(* Logix 5000 project; controller Thurs_Lab2 vendor 1 type 14 code 156 rev 30.11; software revision 30.00; part 4 of 5 *)
(* tags used below, declared in another part *)
   STEP1 : SFC_STEP;
   A_VFD_RUN : BOOL;
   AUTO : BOOL;
   AVERAGE : DINT;
   BLUE_STACK_LITE : BOOL;
   COUNTER : COUNTER;
   CYCLE_COUNT : COUNTER;
   CYCLE_TIME : TIMER;
   CYL1_EXT_4_SORTING : BOOL;
   CYL1_EXT_PX : BOOL;
   CYL1_RET_4_SORTING : BOOL;
   CYL1_RET_PX : BOOL;
   CYL2_EXT_4_SORTING : BOOL;
   CYL2_EXT_PX : BOOL;
   CYL3_EXT : BOOL;
   CYL3_RET : BOOL;
   CYL4_EXT : BOOL;
   CYLINDER1_EXTEND : BOOL;
   CYLINDER1_RETRACT : BOOL;
   CYLINDER2_EXTEND : BOOL;
   CYLINDERSTATUS : DINT;
   DEEP : COUNTER;
   DELAY_PE_INPUT_PSW : TIMER;
   DELAY_PE_INPUT_STATE : TIMER;
   DRILL3 : DRILL3;
   DRILL4 : DRILL4;
   EXTEND : TIMER;
   FAULT : BOOL;
   FAULT_COUNTER : COUNTER;
   GREEN_STACK_LITE : BOOL;
   LAST_CYCLE_COUNT : COUNTER;
   LAST_CYCLE_TIME : DINT;
   MOTOR_WHEEL : BOOL;
   MOTOR_WHEEL_PE : BOOL;
   ONE_SHOT_PSW0 : BOOL;
   ONE_SHOT_PSW1 : BOOL;
   ONE_SHOT_STATE0 : BOOL;
   ONE_SHOT_STATE1 : BOOL;
   OP3_STOP : BOOL;
   OP4_STOP : BOOL;
   OP7_STOP : BOOL;
   OPERATION : DINT;
   OPERATION_7_OVER : BOOL;
   OPERATION_7_REJECT : BOOL;
   OPERATION_7_UNDER : BOOL;
   OPERATION_DONE : DINT;
   OPERATION_OFF : DINT;
   OUTPUT : INT;
   PARTS : COUNTER;
   PARTS_COUNT_TOTALIZER : COUNTER;
   PB1 : BOOL;
   PB1_ON : DINT;
   PILOT_LIGHT_0 : BOOL;
   PILOT_LIGHT_1 : BOOL;
   PILOT_LIGHT_2 : BOOL;
   PILOT_LIGHT_3 : BOOL;
   PILOT_LIGHT_4 : BOOL;
   PILOT_LIGHT_5 : BOOL;
   PREVENT_FAULT_7 : DINT;
   PRODUCTION_ONE_SHOT : BOOL;
   PV_FAULT_COUNT_RESET : BOOL;
   PV_FAULT_RESET : BOOL;
   PV_LAST_CYCLE_TIME1 : DINT;
   PV_LAST_CYCLE_TIME2 : DINT;
   PV_LAST_CYCLE_TIME3 : DINT;
   PV_LAST_CYCLE_TIME4 : DINT;
   PV_LAST_CYCLE_TIME5 : DINT;
   PV_MAX_DEPTH : DINT;
   PV_MIN_DEPTH : DINT;
   PV_PARTS_COUNT_RESET : BOOL;
   PV_RESET : BOOL;
   RED_STACK_LITE : BOOL;
   RESET : BOOL;
   REVOLUTIONS : COUNTER;
   RUN_DC_MOTOR : BOOL;
   SEQ_A_TO_D_COMPLETE : BOOL;
   SEQ_EN : BOOL;
   SETSPEED7 : DINT;
   SHALLOW : COUNTER;
   SORT_SEQ_FOR_REJECT : DINT;
   STA : DINT;
   START_SIGNAL : BOOL;
   STATE : DINT;
   STEP : DINT;
   T : DINT;
   Timer : TIMER;
   TIMER_CELL_DONE : TIMER;
   TO_CELL : TO_CELL;
   TOO_DEEP : BOOL;
   TOO_SHALLOW : BOOL;
   TRANSFER7 : TIMER;
   UP2SPEED7 : TIMER;
   WHITE_STACK_LITE : BOOL;
   YELLOW_STACK_LITE : BOOL;
   ZEROSPEED7 : TIMER;
(* MainProgram, continued *)

ROUTINE OP3_DRILL_PSW   (* ladder *)
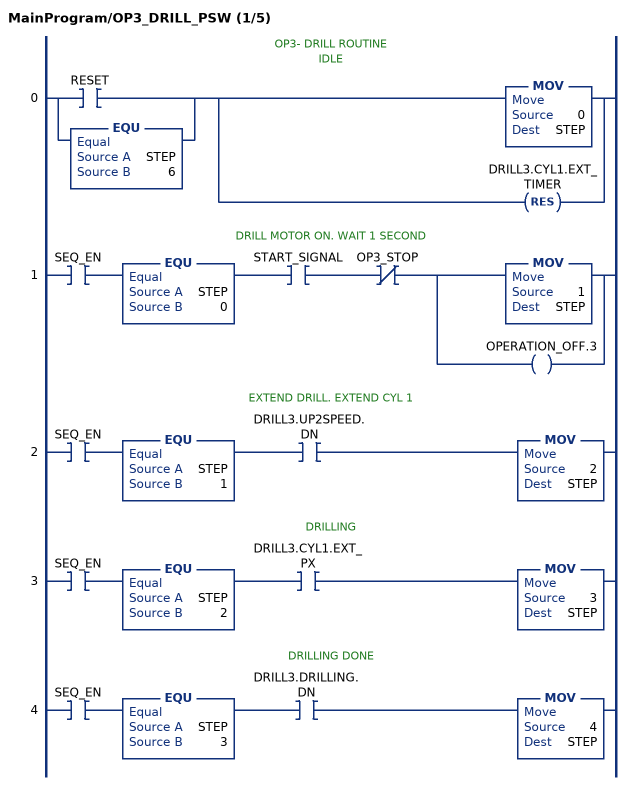
   // OP3- DRILL ROUTINE
   // IDLE
   0: [XIC(RESET) ,EQU(STEP,6) ][MOV(0,STEP) ,RES(DRILL3.CYL1.EXT_TIMER) ];
   // DRILL MOTOR ON. WAIT 1 SECOND
   1: XIC(SEQ_EN)EQU(STEP,0)XIC(START_SIGNAL)XIO(OP3_STOP)[MOV(1,STEP) ,OTE(OPERATION_OFF.3) ];
   // EXTEND DRILL. EXTEND CYL 1
   2: XIC(SEQ_EN)EQU(STEP,1)XIC(DRILL3.UP2SPEED.DN)MOV(2,STEP);
   // DRILLING
   3: XIC(SEQ_EN)EQU(STEP,2)XIC(DRILL3.CYL1.EXT_PX)MOV(3,STEP);
   // DRILLING DONE
   4: XIC(SEQ_EN)EQU(STEP,3)XIC(DRILL3.DRILLING.DN)MOV(4,STEP);
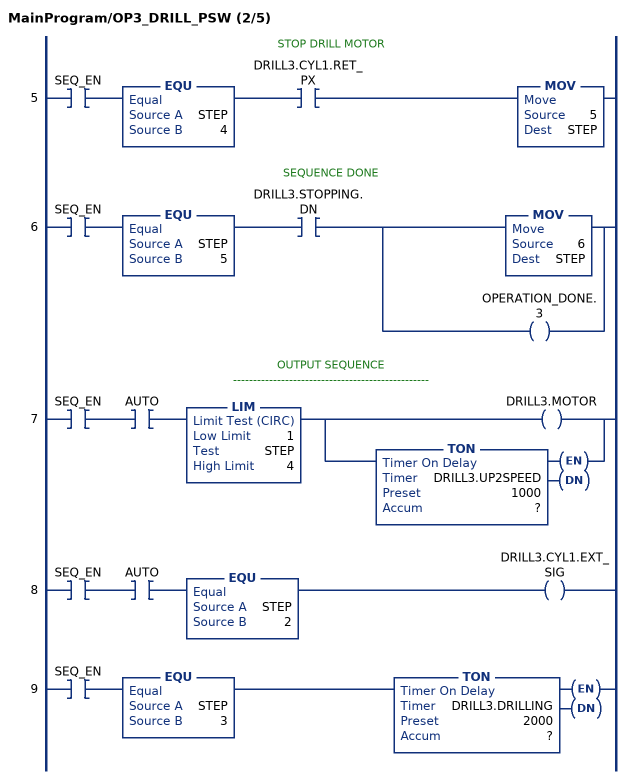
   // STOP DRILL MOTOR
   5: XIC(SEQ_EN)EQU(STEP,4)XIC(DRILL3.CYL1.RET_PX)MOV(5,STEP);
   // SEQUENCE DONE
   6: XIC(SEQ_EN)EQU(STEP,5)XIC(DRILL3.STOPPING.DN)[MOV(6,STEP) ,OTE(OPERATION_DONE.3) ];
   // OUTPUT SEQUENCE
   // -------------------------------------------------
   7: XIC(SEQ_EN)XIC(AUTO)LIM(1,STEP,4)[OTE(DRILL3.MOTOR) ,TON(DRILL3.UP2SPEED,?,?) ];
   8: XIC(SEQ_EN)XIC(AUTO)EQU(STEP,2)OTE(DRILL3.CYL1.EXT_SIG);
   9: XIC(SEQ_EN)EQU(STEP,3)TON(DRILL3.DRILLING,?,?);
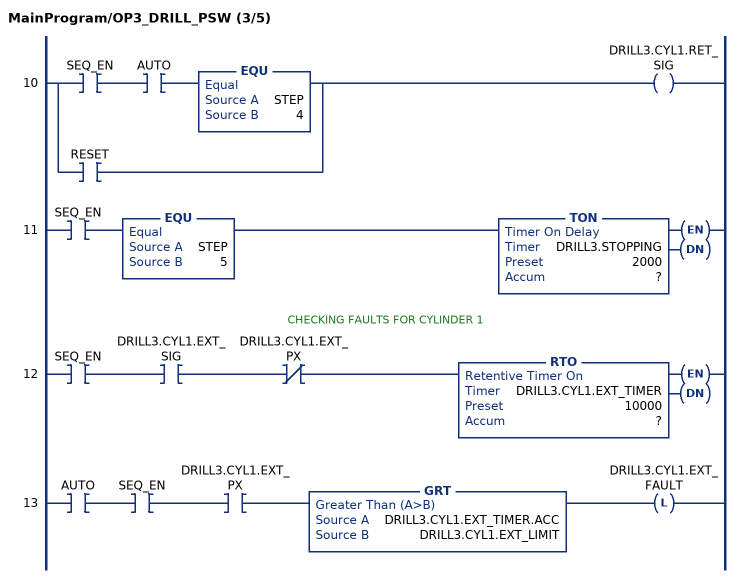
   10: [XIC(SEQ_EN) XIC(AUTO) EQU(STEP,4) ,XIC(RESET) ]OTE(DRILL3.CYL1.RET_SIG);
   11: XIC(SEQ_EN)EQU(STEP,5)TON(DRILL3.STOPPING,?,?);
   // CHECKING FAULTS FOR CYLINDER 1
   12: XIC(SEQ_EN)XIC(DRILL3.CYL1.EXT_SIG)XIO(DRILL3.CYL1.EXT_PX)RTO(DRILL3.CYL1.EXT_TIMER,?,?);
   13: XIC(AUTO)XIC(SEQ_EN)XIC(DRILL3.CYL1.EXT_PX)GRT(DRILL3.CYL1.EXT_TIMER.ACC,DRILL3.CYL1.EXT_LIMIT)OTL(DRILL3.CYL1.EXT_FAULT);
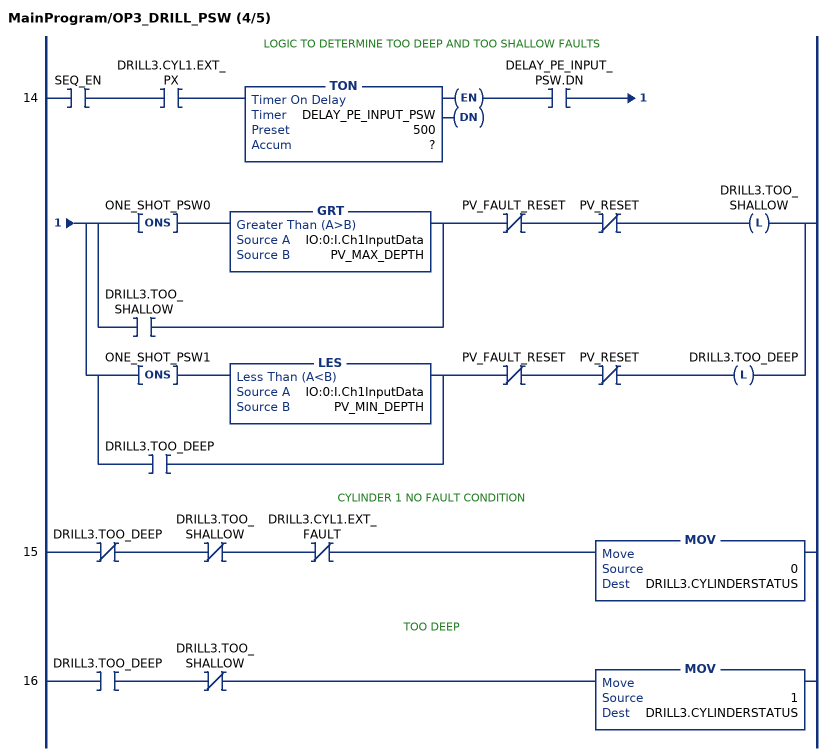
   // LOGIC TO DETERMINE TOO DEEP AND TOO SHALLOW FAULTS
   14: XIC(SEQ_EN)XIC(DRILL3.CYL1.EXT_PX)TON(DELAY_PE_INPUT_PSW,?,?)XIC(DELAY_PE_INPUT_PSW.DN)[[ONS(ONE_SHOT_PSW0) GRT(IO:0:I.Ch1InputData,PV_MAX_DEPTH) ,XIC(DRILL3.TOO_SHALLOW) ] XIO(PV_FAULT_RESET) XIO(PV_RESET) OTL(DRILL3.TOO_SHALLOW) ,[ONS(ONE_SHOT_PSW1) LES(IO:0:I.Ch1InputData,PV_MIN_DEPTH) ,XIC(DRILL3.TOO_DEEP) ] XIO(PV_FAULT_RESET) XIO(PV_RESET) OTL(DRILL3.TOO_DEEP) ];
   // CYLINDER 1 NO FAULT CONDITION
   15: XIO(DRILL3.TOO_DEEP)XIO(DRILL3.TOO_SHALLOW)XIO(DRILL3.CYL1.EXT_FAULT)MOV(0,DRILL3.CYLINDERSTATUS);
   // TOO DEEP
   16: XIC(DRILL3.TOO_DEEP)XIO(DRILL3.TOO_SHALLOW)MOV(1,DRILL3.CYLINDERSTATUS);
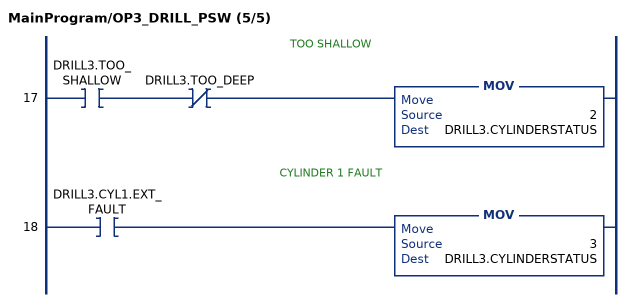
   // TOO SHALLOW
   17: XIC(DRILL3.TOO_SHALLOW)XIO(DRILL3.TOO_DEEP)MOV(2,DRILL3.CYLINDERSTATUS);
   // CYLINDER 1 FAULT
   18: XIC(DRILL3.CYL1.EXT_FAULT)MOV(3,DRILL3.CYLINDERSTATUS);
END_ROUTINE

ROUTINE OP4_DRILL_STATE   (* ladder *)
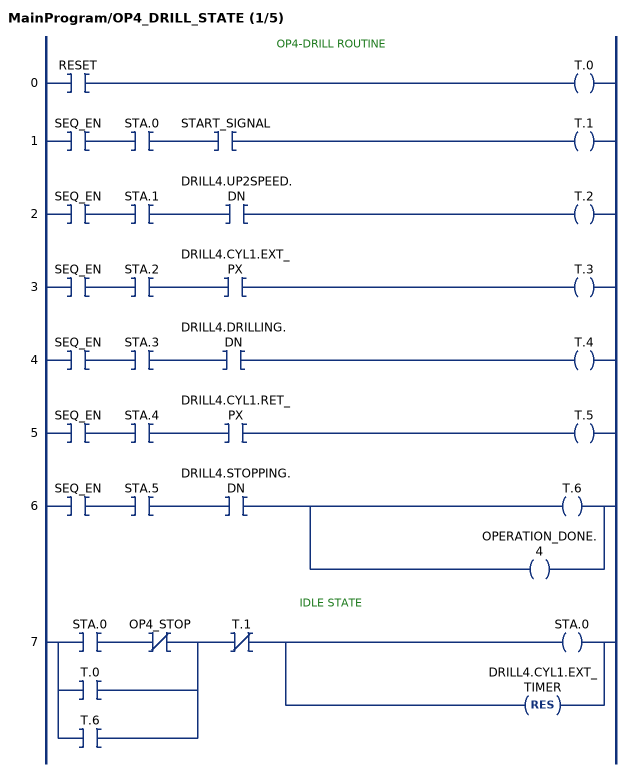
   // OP4-DRILL ROUTINE
   0: XIC(RESET)OTE(T.0);
   1: XIC(SEQ_EN)XIC(STA.0)XIC(START_SIGNAL)OTE(T.1);
   2: XIC(SEQ_EN)XIC(STA.1)XIC(DRILL4.UP2SPEED.DN)OTE(T.2);
   3: XIC(SEQ_EN)XIC(STA.2)XIC(DRILL4.CYL1.EXT_PX)OTE(T.3);
   4: XIC(SEQ_EN)XIC(STA.3)XIC(DRILL4.DRILLING.DN)OTE(T.4);
   5: XIC(SEQ_EN)XIC(STA.4)XIC(DRILL4.CYL1.RET_PX)OTE(T.5);
   6: XIC(SEQ_EN)XIC(STA.5)XIC(DRILL4.STOPPING.DN)[OTE(T.6) ,OTE(OPERATION_DONE.4) ];
   // IDLE STATE
   7: [XIC(STA.0) XIO(OP4_STOP) ,XIC(T.0) ,XIC(T.6) ]XIO(T.1)[OTE(STA.0) ,RES(DRILL4.CYL1.EXT_TIMER) ];
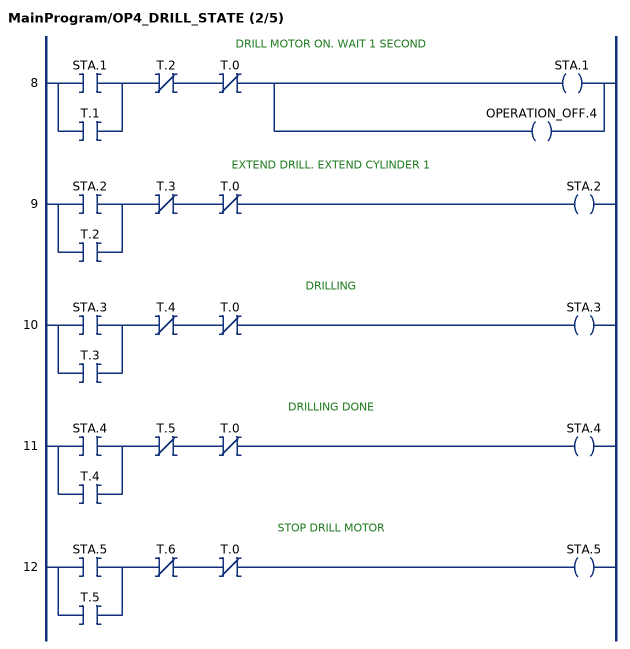
   // DRILL MOTOR ON. WAIT 1 SECOND
   8: [XIC(STA.1) ,XIC(T.1) ]XIO(T.2)XIO(T.0)[OTE(STA.1) ,OTE(OPERATION_OFF.4) ];
   // EXTEND DRILL. EXTEND CYLINDER 1
   9: [XIC(STA.2) ,XIC(T.2) ]XIO(T.3)XIO(T.0)OTE(STA.2);
   // DRILLING
   10: [XIC(STA.3) ,XIC(T.3) ]XIO(T.4)XIO(T.0)OTE(STA.3);
   // DRILLING DONE
   11: [XIC(STA.4) ,XIC(T.4) ]XIO(T.5)XIO(T.0)OTE(STA.4);
   // STOP DRILL MOTOR
   12: [XIC(STA.5) ,XIC(T.5) ]XIO(T.6)XIO(T.0)OTE(STA.5);
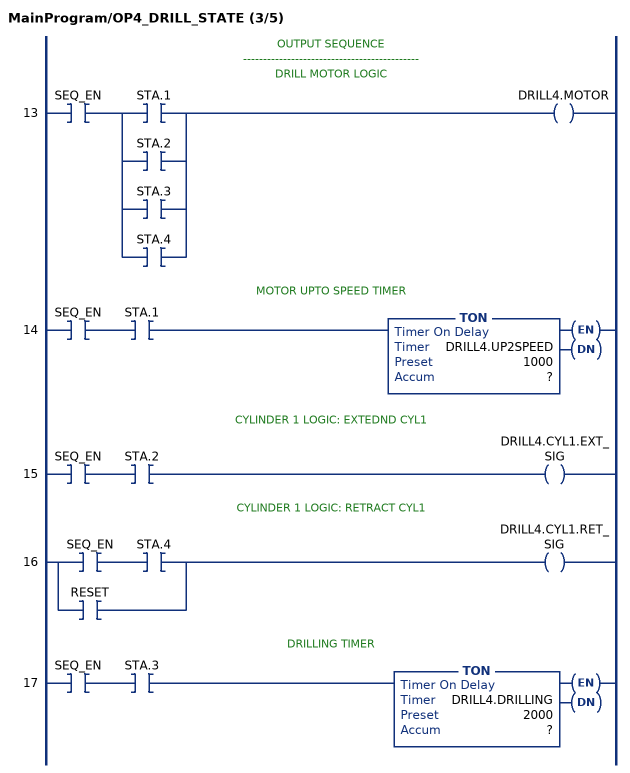
   // OUTPUT SEQUENCE
   // --------------------------------------------
   // DRILL MOTOR LOGIC
   13: XIC(SEQ_EN)[XIC(STA.1) ,XIC(STA.2) ,XIC(STA.3) ,XIC(STA.4) ]OTE(DRILL4.MOTOR);
   // MOTOR UPTO SPEED TIMER
   14: XIC(SEQ_EN)XIC(STA.1)TON(DRILL4.UP2SPEED,?,?);
   // CYLINDER 1 LOGIC: EXTEDND CYL1
   15: XIC(SEQ_EN)XIC(STA.2)OTE(DRILL4.CYL1.EXT_SIG);
   // CYLINDER 1 LOGIC: RETRACT CYL1
   16: [XIC(SEQ_EN) XIC(STA.4) ,XIC(RESET) ]OTE(DRILL4.CYL1.RET_SIG);
   // DRILLING TIMER
   17: XIC(SEQ_EN)XIC(STA.3)TON(DRILL4.DRILLING,?,?);
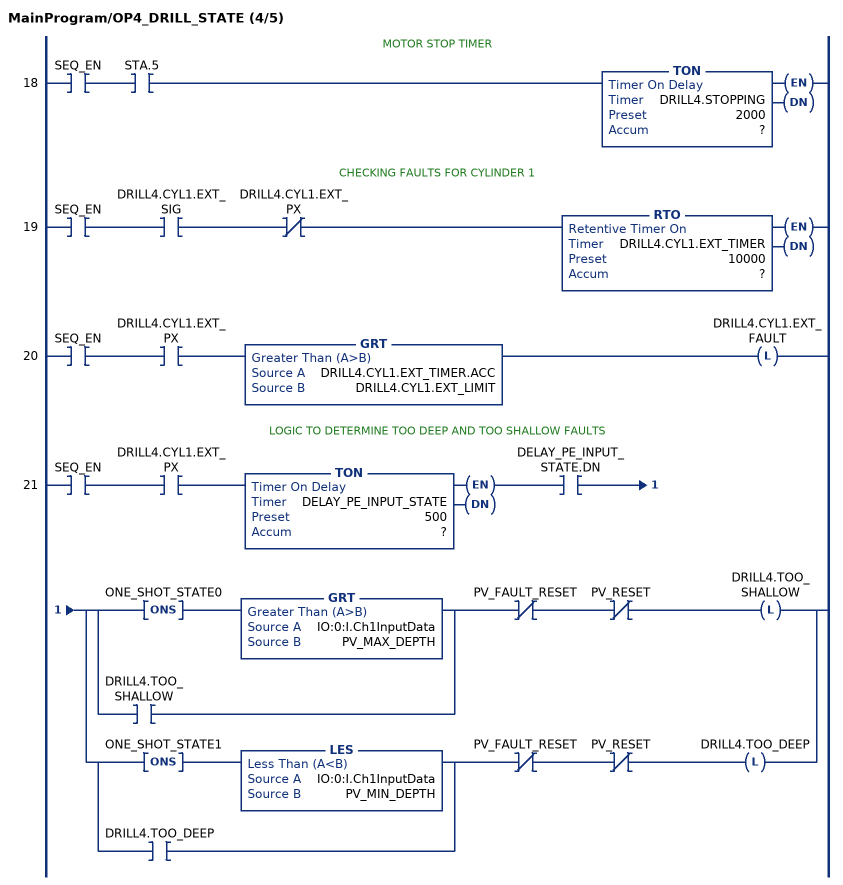
   // MOTOR STOP TIMER
   18: XIC(SEQ_EN)XIC(STA.5)TON(DRILL4.STOPPING,?,?);
   // CHECKING FAULTS FOR CYLINDER 1
   19: XIC(SEQ_EN)XIC(DRILL4.CYL1.EXT_SIG)XIO(DRILL4.CYL1.EXT_PX)RTO(DRILL4.CYL1.EXT_TIMER,?,?);
   20: XIC(SEQ_EN)XIC(DRILL4.CYL1.EXT_PX)GRT(DRILL4.CYL1.EXT_TIMER.ACC,DRILL4.CYL1.EXT_LIMIT)OTL(DRILL4.CYL1.EXT_FAULT);
   // LOGIC TO DETERMINE TOO DEEP AND TOO SHALLOW FAULTS
   21: XIC(SEQ_EN)XIC(DRILL4.CYL1.EXT_PX)TON(DELAY_PE_INPUT_STATE,?,?)XIC(DELAY_PE_INPUT_STATE.DN)[[ONS(ONE_SHOT_STATE0) GRT(IO:0:I.Ch1InputData,PV_MAX_DEPTH) ,XIC(DRILL4.TOO_SHALLOW) ] XIO(PV_FAULT_RESET) XIO(PV_RESET) OTL(DRILL4.TOO_SHALLOW) ,[ONS(ONE_SHOT_STATE1) LES(IO:0:I.Ch1InputData,PV_MIN_DEPTH) ,XIC(DRILL4.TOO_DEEP) ] XIO(PV_FAULT_RESET) XIO(PV_RESET) OTL(DRILL4.TOO_DEEP) ];
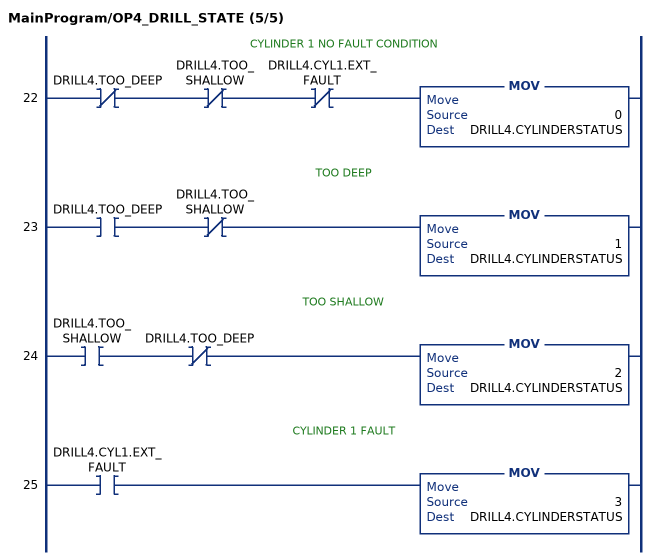
   // CYLINDER 1 NO FAULT CONDITION
   22: XIO(DRILL4.TOO_DEEP)XIO(DRILL4.TOO_SHALLOW)XIO(DRILL4.CYL1.EXT_FAULT)MOV(0,DRILL4.CYLINDERSTATUS);
   // TOO DEEP
   23: XIC(DRILL4.TOO_DEEP)XIO(DRILL4.TOO_SHALLOW)MOV(1,DRILL4.CYLINDERSTATUS);
   // TOO SHALLOW
   24: XIC(DRILL4.TOO_SHALLOW)XIO(DRILL4.TOO_DEEP)MOV(2,DRILL4.CYLINDERSTATUS);
   // CYLINDER 1 FAULT
   25: XIC(DRILL4.CYL1.EXT_FAULT)MOV(3,DRILL4.CYLINDERSTATUS);
END_ROUTINE

ROUTINE OUTPUT_BUFFERING   (* function block diagram *)
   SHEET 1
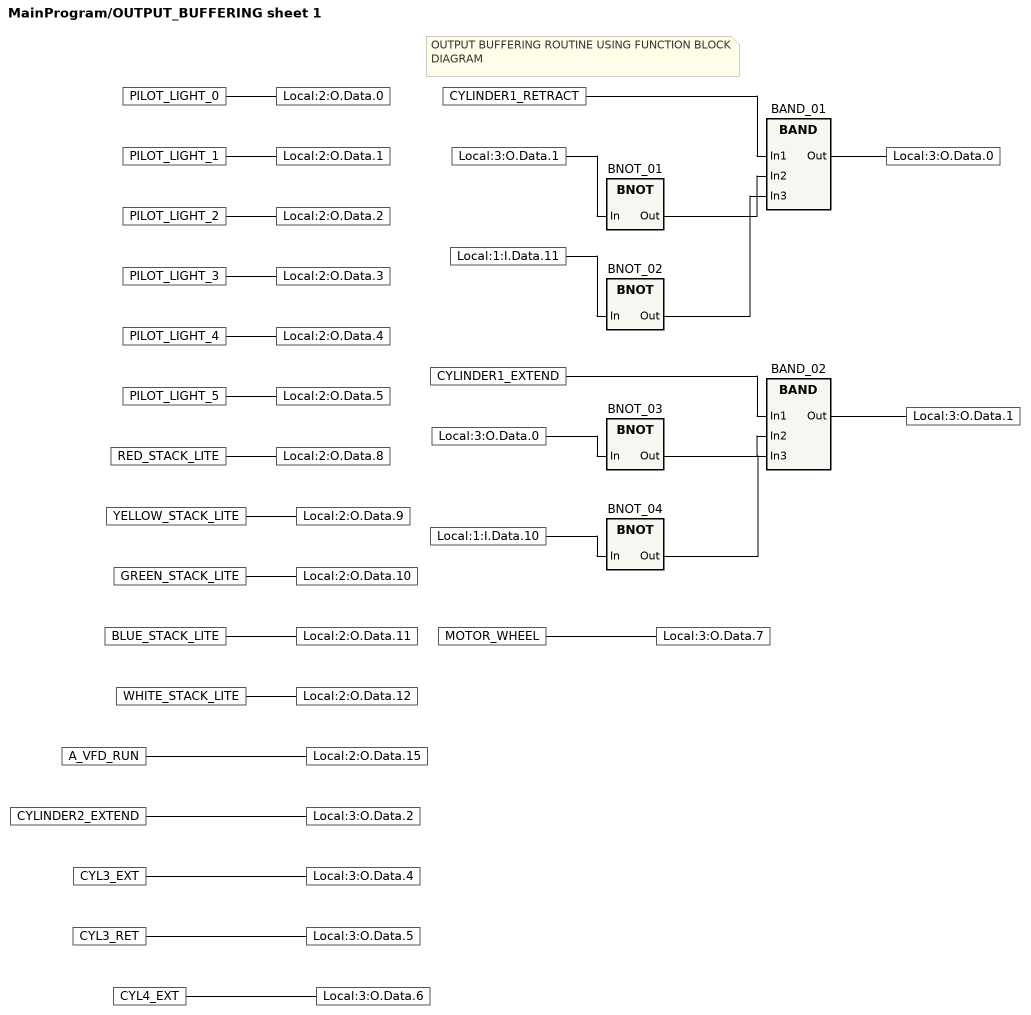
   // OUTPUT BUFFERING ROUTINE USING FUNCTION BLOCK DIAGRAM
   Local:2:O.Data.0 := PILOT_LIGHT_0;
   Local:2:O.Data.1 := PILOT_LIGHT_1;
   Local:2:O.Data.2 := PILOT_LIGHT_2;
   Local:2:O.Data.3 := PILOT_LIGHT_3;
   Local:2:O.Data.4 := PILOT_LIGHT_4;
   Local:2:O.Data.5 := PILOT_LIGHT_5;
   Local:2:O.Data.8 := RED_STACK_LITE;
   Local:2:O.Data.9 := YELLOW_STACK_LITE;
   Local:2:O.Data.10 := GREEN_STACK_LITE;
   Local:2:O.Data.11 := BLUE_STACK_LITE;
   Local:2:O.Data.12 := WHITE_STACK_LITE;
   Local:2:O.Data.15 := A_VFD_RUN;
   Local:3:O.Data.2 := CYLINDER2_EXTEND;
   Local:3:O.Data.4 := CYL3_EXT;
   Local:3:O.Data.5 := CYL3_RET;
   Local:3:O.Data.6 := CYL4_EXT;
   BNOT_01 : BNOT(In := Local:3:O.Data.1);
   BNOT_02 : BNOT(In := Local:1:I.Data.11);
   BNOT_03 : BNOT(In := Local:3:O.Data.0);
   BNOT_04 : BNOT(In := Local:1:I.Data.10);
   Local:3:O.Data.7 := MOTOR_WHEEL;
   BAND_01 : BAND(In1 := CYLINDER1_RETRACT, In2 := BNOT_01.Out, In3 := BNOT_02.Out);
   BAND_02 : BAND(In1 := CYLINDER1_EXTEND, In2 := BNOT_03.Out, In3 := BNOT_04.Out);
   Local:3:O.Data.0 := BAND_01.Out;
   Local:3:O.Data.1 := BAND_02.Out;
END_ROUTINE

ROUTINE PRODUCTION   (* ladder *)
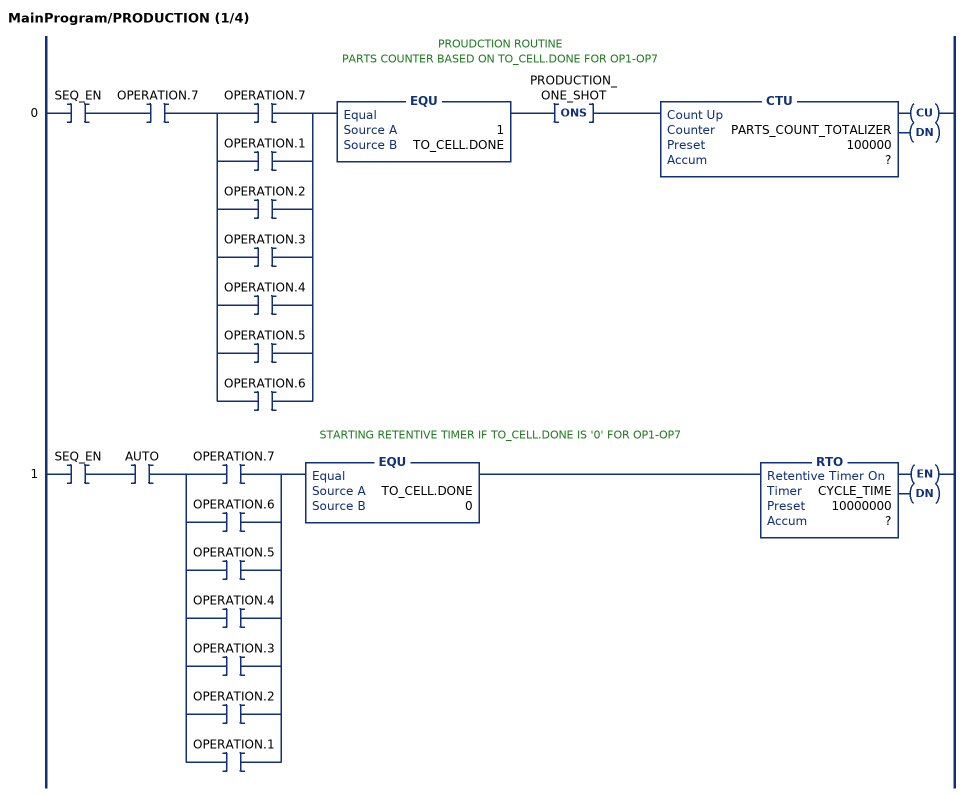
   // PROUDCTION ROUTINE
   // PARTS COUNTER BASED ON TO_CELL.DONE FOR OP1-OP7
   0: XIC(SEQ_EN)XIC(OPERATION.7)[XIC(OPERATION.7) ,XIC(OPERATION.1) ,XIC(OPERATION.2) ,XIC(OPERATION.3) ,XIC(OPERATION.4) ,XIC(OPERATION.5) ,XIC(OPERATION.6) ]EQU(1,TO_CELL.DONE)ONS(PRODUCTION_ONE_SHOT)CTU(PARTS_COUNT_TOTALIZER,?,?);
   // STARTING RETENTIVE TIMER IF TO_CELL.DONE IS '0' FOR OP1-OP7
   1: XIC(SEQ_EN)XIC(AUTO)[XIC(OPERATION.7) ,XIC(OPERATION.6) ,XIC(OPERATION.5) ,XIC(OPERATION.4) ,XIC(OPERATION.3) ,XIC(OPERATION.2) ,XIC(OPERATION.1) ]EQU(TO_CELL.DONE,0)RTO(CYCLE_TIME,?,?);
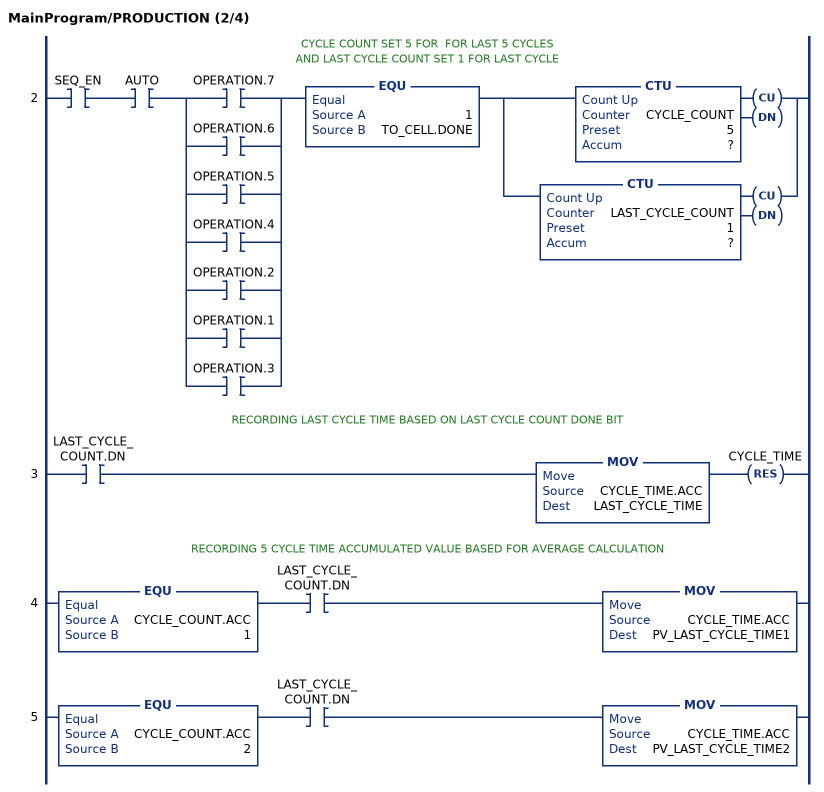
   // CYCLE COUNT SET 5 FOR  FOR LAST 5 CYCLES
   // AND LAST CYCLE COUNT SET 1 FOR LAST CYCLE
   2: XIC(SEQ_EN)XIC(AUTO)[XIC(OPERATION.7) ,XIC(OPERATION.6) ,XIC(OPERATION.5) ,XIC(OPERATION.4) ,XIC(OPERATION.2) ,XIC(OPERATION.1) ,XIC(OPERATION.3) ]EQU(1,TO_CELL.DONE)[CTU(CYCLE_COUNT,?,?) ,CTU(LAST_CYCLE_COUNT,?,?) ];
   // RECORDING LAST CYCLE TIME BASED ON LAST CYCLE COUNT DONE BIT
   3: XIC(LAST_CYCLE_COUNT.DN)MOV(CYCLE_TIME.ACC,LAST_CYCLE_TIME)RES(CYCLE_TIME);
   // RECORDING 5 CYCLE TIME ACCUMULATED VALUE BASED FOR AVERAGE CALCULATION
   4: EQU(CYCLE_COUNT.ACC,1)XIC(LAST_CYCLE_COUNT.DN)MOV(CYCLE_TIME.ACC,PV_LAST_CYCLE_TIME1);
   5: EQU(CYCLE_COUNT.ACC,2)XIC(LAST_CYCLE_COUNT.DN)MOV(CYCLE_TIME.ACC,PV_LAST_CYCLE_TIME2);
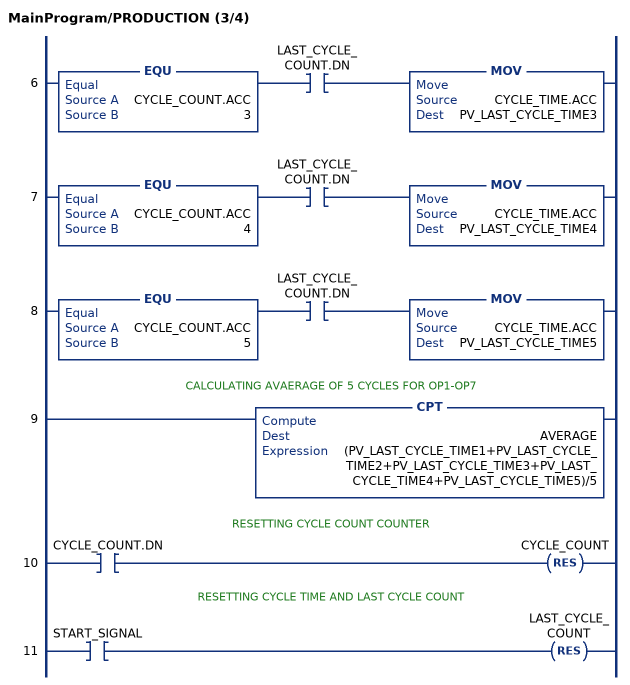
   6: EQU(CYCLE_COUNT.ACC,3)XIC(LAST_CYCLE_COUNT.DN)MOV(CYCLE_TIME.ACC,PV_LAST_CYCLE_TIME3);
   7: EQU(CYCLE_COUNT.ACC,4)XIC(LAST_CYCLE_COUNT.DN)MOV(CYCLE_TIME.ACC,PV_LAST_CYCLE_TIME4);
   8: EQU(CYCLE_COUNT.ACC,5)XIC(LAST_CYCLE_COUNT.DN)MOV(CYCLE_TIME.ACC,PV_LAST_CYCLE_TIME5);
   // CALCULATING AVAERAGE OF 5 CYCLES FOR OP1-OP7
   9: CPT(AVERAGE,(PV_LAST_CYCLE_TIME1+PV_LAST_CYCLE_TIME2+PV_LAST_CYCLE_TIME3+PV_LAST_CYCLE_TIME4+PV_LAST_CYCLE_TIME5)/5);
   // RESETTING CYCLE COUNT COUNTER
   10: XIC(CYCLE_COUNT.DN)RES(CYCLE_COUNT);
   // RESETTING CYCLE TIME AND LAST CYCLE COUNT
   11: XIC(START_SIGNAL)RES(LAST_CYCLE_COUNT);
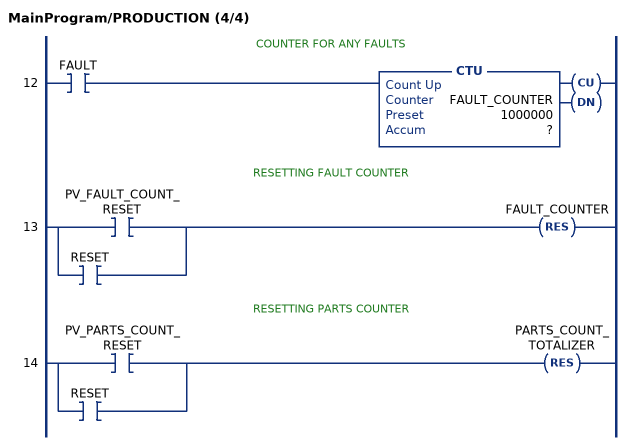
   // COUNTER FOR ANY FAULTS
   12: XIC(FAULT)CTU(FAULT_COUNTER,?,?);
   // RESETTING FAULT COUNTER
   13: [XIC(PV_FAULT_COUNT_RESET) ,XIC(RESET) ]RES(FAULT_COUNTER);
   // RESETTING PARTS COUNTER
   14: [XIC(PV_PARTS_COUNT_RESET) ,XIC(RESET) ]RES(PARTS_COUNT_TOTALIZER);
END_ROUTINE

ROUTINE SORT   (* ladder *)
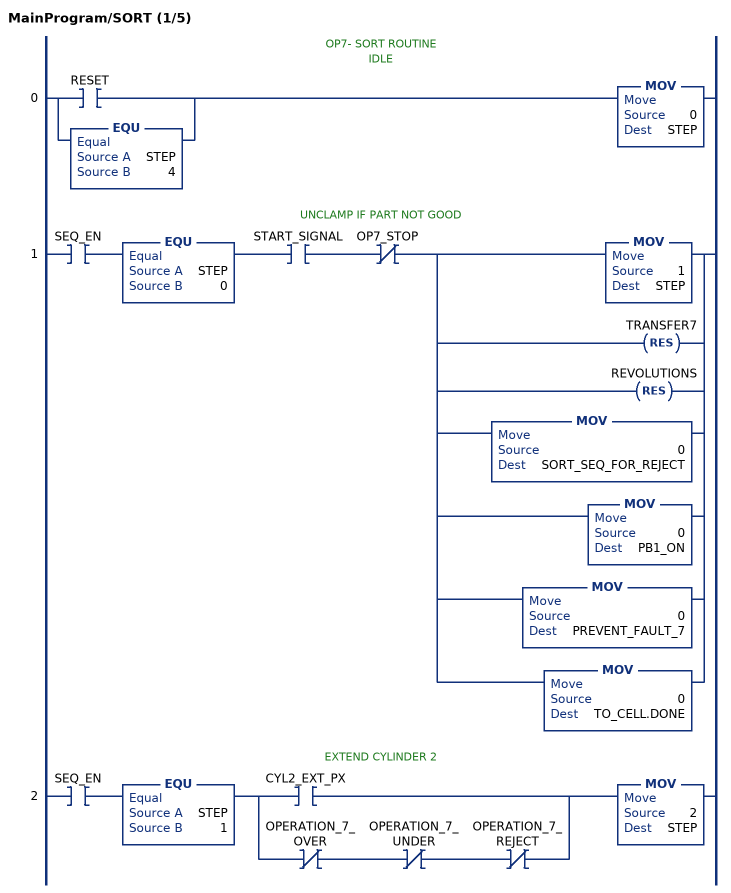
   // OP7- SORT ROUTINE
   // IDLE
   0: [XIC(RESET) ,EQU(STEP,4) ]MOV(0,STEP);
   // UNCLAMP IF PART NOT GOOD
   1: XIC(SEQ_EN)EQU(STEP,0)XIC(START_SIGNAL)XIO(OP7_STOP)[MOV(1,STEP) ,RES(TRANSFER7) ,RES(REVOLUTIONS) ,MOV(0,SORT_SEQ_FOR_REJECT) ,MOV(0,PB1_ON) ,MOV(0,PREVENT_FAULT_7) ,MOV(0,TO_CELL.DONE) ];
   // EXTEND CYLINDER 2
   2: XIC(SEQ_EN)EQU(STEP,1)[XIC(CYL2_EXT_PX) ,XIO(OPERATION_7_OVER) XIO(OPERATION_7_UNDER) XIO(OPERATION_7_REJECT) ]MOV(2,STEP);
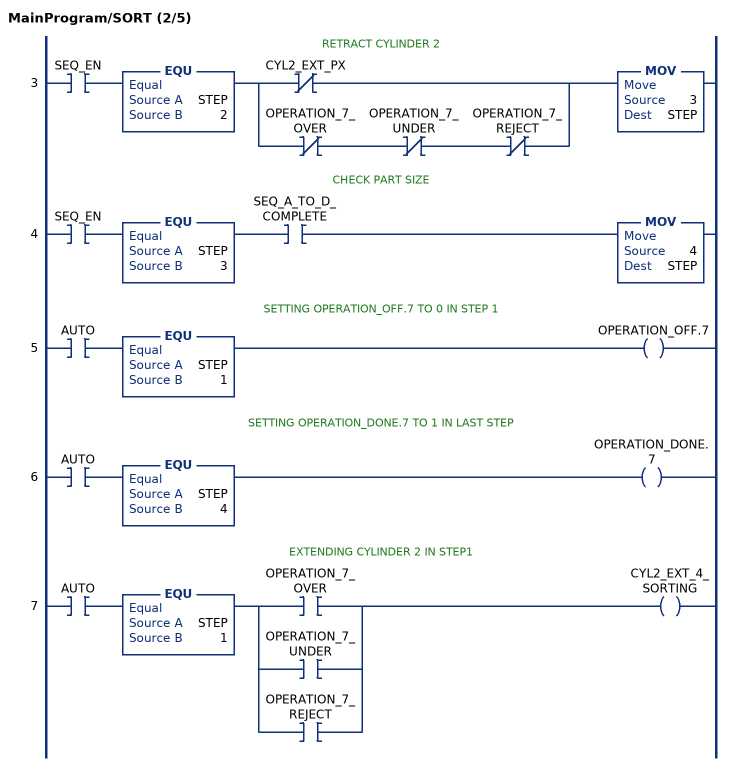
   // RETRACT CYLINDER 2
   3: XIC(SEQ_EN)EQU(STEP,2)[XIO(CYL2_EXT_PX) ,XIO(OPERATION_7_OVER) XIO(OPERATION_7_UNDER) XIO(OPERATION_7_REJECT) ]MOV(3,STEP);
   // CHECK PART SIZE
   4: XIC(SEQ_EN)EQU(STEP,3)XIC(SEQ_A_TO_D_COMPLETE)MOV(4,STEP);
   // SETTING OPERATION_OFF.7 TO 0 IN STEP 1
   5: XIC(AUTO)EQU(STEP,1)OTE(OPERATION_OFF.7);
   // SETTING OPERATION_DONE.7 TO 1 IN LAST STEP
   6: XIC(AUTO)EQU(STEP,4)OTE(OPERATION_DONE.7);
   // EXTENDING CYLINDER 2 IN STEP1
   7: XIC(AUTO)EQU(STEP,1)[XIC(OPERATION_7_OVER) ,XIC(OPERATION_7_UNDER) ,XIC(OPERATION_7_REJECT) ]OTE(CYL2_EXT_4_SORTING);
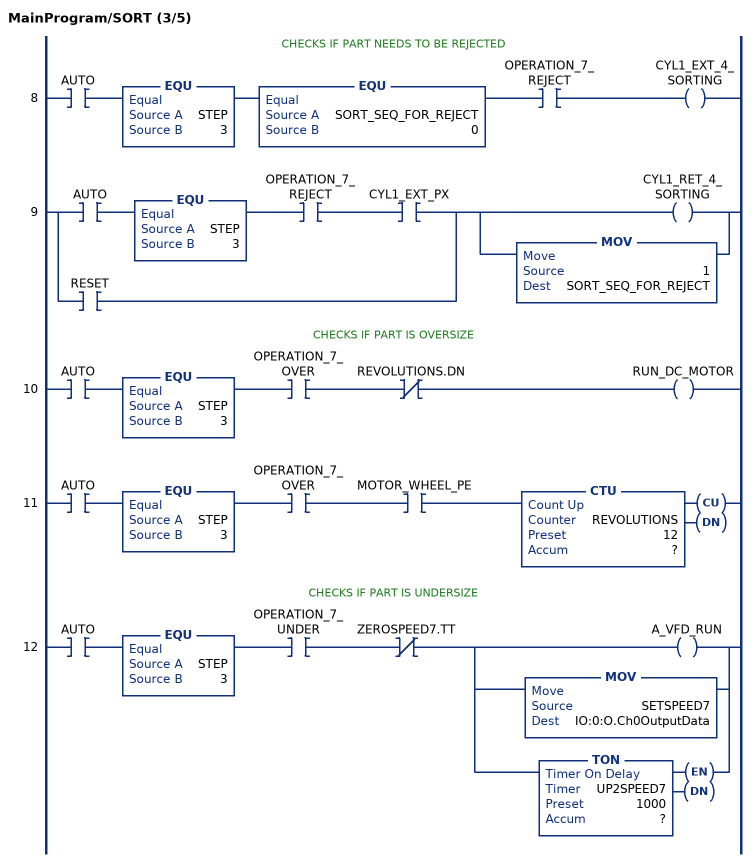
   // CHECKS IF PART NEEDS TO BE REJECTED
   8: XIC(AUTO)EQU(STEP,3)EQU(SORT_SEQ_FOR_REJECT,0)XIC(OPERATION_7_REJECT)OTE(CYL1_EXT_4_SORTING);
   9: [XIC(AUTO) EQU(STEP,3) XIC(OPERATION_7_REJECT) XIC(CYL1_EXT_PX) ,XIC(RESET) ][OTE(CYL1_RET_4_SORTING) ,MOV(1,SORT_SEQ_FOR_REJECT) ];
   // CHECKS IF PART IS OVERSIZE
   10: XIC(AUTO)EQU(STEP,3)XIC(OPERATION_7_OVER)XIO(REVOLUTIONS.DN)OTE(RUN_DC_MOTOR);
   11: XIC(AUTO)EQU(STEP,3)XIC(OPERATION_7_OVER)XIC(MOTOR_WHEEL_PE)CTU(REVOLUTIONS,?,?);
   // CHECKS IF PART IS UNDERSIZE
   12: XIC(AUTO)EQU(STEP,3)XIC(OPERATION_7_UNDER)XIO(ZEROSPEED7.TT)[OTE(A_VFD_RUN) ,MOV(SETSPEED7,IO:0:O.Ch0OutputData) ,TON(UP2SPEED7,?,?) ];
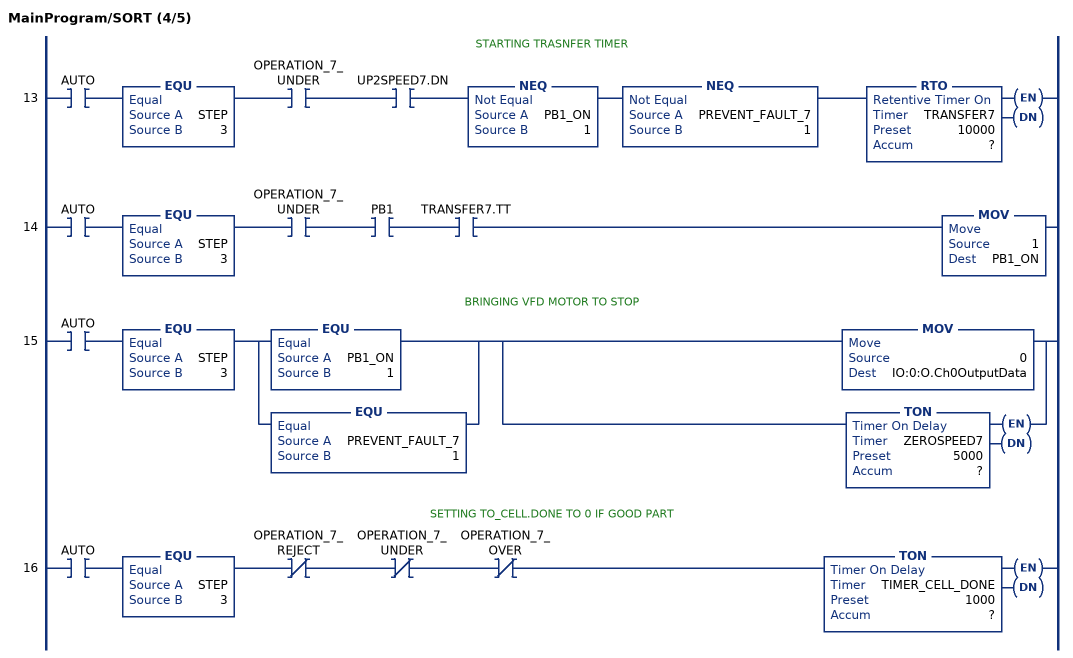
   // STARTING TRASNFER TIMER
   13: XIC(AUTO)EQU(STEP,3)XIC(OPERATION_7_UNDER)XIC(UP2SPEED7.DN)NEQ(PB1_ON,1)NEQ(PREVENT_FAULT_7,1)RTO(TRANSFER7,?,?);
   14: XIC(AUTO)EQU(STEP,3)XIC(OPERATION_7_UNDER)XIC(PB1)XIC(TRANSFER7.TT)MOV(1,PB1_ON);
   // BRINGING VFD MOTOR TO STOP
   15: XIC(AUTO)EQU(STEP,3)[EQU(PB1_ON,1) ,EQU(PREVENT_FAULT_7,1) ][MOV(0,IO:0:O.Ch0OutputData) ,TON(ZEROSPEED7,?,?) ];
   // SETTING TO_CELL.DONE TO 0 IF GOOD PART
   16: XIC(AUTO)EQU(STEP,3)XIO(OPERATION_7_REJECT)XIO(OPERATION_7_UNDER)XIO(OPERATION_7_OVER)TON(TIMER_CELL_DONE,?,?);
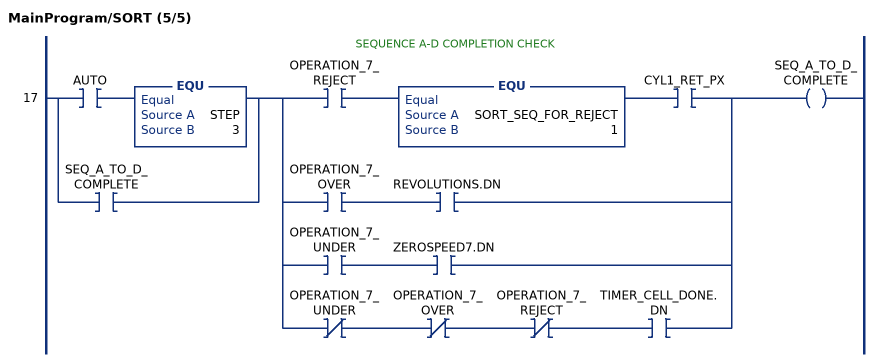
   // SEQUENCE A-D COMPLETION CHECK
   17: [XIC(AUTO) EQU(STEP,3) ,XIC(SEQ_A_TO_D_COMPLETE) ][XIC(OPERATION_7_REJECT) EQU(SORT_SEQ_FOR_REJECT,1) XIC(CYL1_RET_PX) ,XIC(OPERATION_7_OVER) XIC(REVOLUTIONS.DN) ,XIC(OPERATION_7_UNDER) XIC(ZEROSPEED7.DN) ,XIO(OPERATION_7_UNDER) XIO(OPERATION_7_OVER) XIO(OPERATION_7_REJECT) XIC(TIMER_CELL_DONE.DN) ]OTE(SEQ_A_TO_D_COMPLETE);
END_ROUTINE
